// calculate horizontal coordinates
eq2hor(
	ra := fRightAscensionCurrent,
	dec := fDeclinationCurrent,
	lon := telescopeConfig.longitude,
	lat := telescopeConfig.latitude,
	JD := fJD,
	alt => fElevationCalc,
	az => fAzimuthCalc,
	ha => fHourAngleCalc);

METHOD _PublishTelemetry : BOOL
VAR_INPUT
END_VAR
fbComm.Publish('telescope', 'dome', 'POSITION.INSTRUMENTAL.RA.OFFSET', LREAL_TO_STRING(fHourAngleOffset));
fbComm.Publish('telescope', 'dome', 'POSITION.INSTRUMENTAL.DEC.OFFSET', LREAL_TO_STRING(fDeclinationOffset));
END_METHOD

PROPERTY DeclinationOffset : LREAL
GET
DeclinationOffset := THIS^.fDeclinationOffset;
END_GET
SET
THIS^.fDeclinationOffset := DeclinationOffset;
END_SET
END_PROPERTY

PROPERTY HourAngleOffset : LREAL
GET
HourAngleOffset := THIS^.fHourAngleOffset;
END_GET
SET
THIS^.fHourAngleOffset := HourAngleOffset;
END_SET
END_PROPERTY

END_FUNCTION_BLOCK
